FUNCTION_BLOCK FB_E2408_Manager
VAR_INPUT
	sendMessage			:ST_Modbus_Send_Frame;
END_VAR
VAR_OUTPUT
	bWriteError			:BOOL; 
	bReadError			:BOOL;
	bSendBufferusFull	:BOOL;
	bConnectError 		: BOOL;
	
	RData_Module_1	:ST_E2408_Data;
	RData_Module_2	:ST_E2408_Data;
	RData_Module_3	:ST_E2408_Data;
	RData_Module_4	:ST_E2408_Data;
	RData_Module_5	:ST_E2408_Data;
	RData_Module_6	:ST_E2408_Data;
END_VAR
VAR
	fbModbus_Master		:ModbusRtuMasterV2_KL6x22B;
	ReconnectTon		:TON;
	DataReadTon			:TON;
	bWriteExecute		:BOOL;
	bReadExecute		:BOOL;
	arrReceivedBuffer 	:ARRAY [0..200] OF WORD;
	arrSendBuffer 		:ARRAY [0..99] OF WORD;
	
	nModbusRead_Start_ADDR	:WORD;
	nModbusWrite_Start_ADDR	:WORD;
	nReadExecuteCount		:UDINT;
		
	fbStructModbusSend:FB_MODBUS_SEND_FIFO;
	stOutput:ST_MODBUS_SEND_FRAME;
	
	nWriteQuantity		:WORD;
	fallEdge			:F_TRIG;
	backCount			: UDINT;
	nCycle				: UDINT;
	ReceivedTime		: UDINT;
	ResendTon			: Ton;
	rinedge				: R_TRIG;
	WriteCount			: INT;
	CheckLoad			: REAL;
	ErrorCount			: INT;
	BufferCount_Zefo	: INT;
	fTrigWriteComplete	: F_TRIG;
	ReReadTon: TON;
	ReReadTrig			: BOOL;
	
	ReadInputRegsBusy		: BOOL;
	ReadInputRegsError		: BOOL;
	WriteSingleRegisterBusy	: BOOL;
	WriteSingleRegisterError: BOOL;
END_VAR

IF  ReadInputRegsError =FALSE THEN
	_Case();
	_CheckSendData();
ELSE
	ReconnectTon(IN:=ReconnectTon.Q=FALSE AND TRUE,pt:=T#1S);
	
	IF ReconnectTon.Q THEN
		
		ErrorCount := ErrorCount +1;
		
		IF ReadInputRegsError = TRUE THEN
			bReadExecute:=NOT bReadExecute;
		END_IF
		
	END_IF
END_IF

_ModbusFunction();
fbStructModbusSend();

bConnectError:= ReadInputRegsError;

ACTION _Case:
IF ReadInputRegsBusy = TRUE OR ReadInputRegsError = TRUE AND bWriteExecute = FALSE AND WriteSingleRegisterBusy = FALSE  THEN
	bReadExecute := FALSE;
	IF ReadInputRegsError = TRUE THEN
		bReadError:=TRUE;
	END_IF
END_IF

(*Copy Data*)
IF (ReadInputRegsBusy = FALSE AND ReadInputRegsError = FALSE)  THEN
	IF (fbModbus_Master.cbRead >0)  (*AND (arrReceivedBuffer[4] <> 0)*) THEN
		
	IF arrReceivedBuffer[4] = 0 THEN
		BufferCount_Zefo:=BufferCount_Zefo +1 ; 
	END_IF

		CASE nReadExecuteCount OF
			1:MEMCPY(ADR(RData_Module_1),ADR(arrReceivedBuffer),SIZEOF(RData_Module_1));
				ReceivedTime :=nCycle;
				nCycle:=0;
			2:MEMCPY(ADR(RData_Module_2),ADR(arrReceivedBuffer),SIZEOF(RData_Module_2));
			3:MEMCPY(ADR(RData_Module_3),ADR(arrReceivedBuffer),SIZEOF(RData_Module_3));
			4:MEMCPY(ADR(RData_Module_4),ADR(arrReceivedBuffer),SIZEOF(RData_Module_4));
			5:MEMCPY(ADR(RData_Module_5),ADR(arrReceivedBuffer),SIZEOF(RData_Module_5));
			6:MEMCPY(ADR(RData_Module_6),ADR(arrReceivedBuffer),SIZEOF(RData_Module_6));
		END_CASE
	END_IF
	
END_IF
nCycle:=nCycle+1;

(*Change Address*)
IF ReadInputRegsBusy = FALSE  AND ReadInputRegsError = FALSE  AND fbStructModbusSend.nBufferCount = 0 AND bWriteExecute = FALSE AND WriteSingleRegisterBusy = FALSE THEN
DataReadTon(IN:=TRUE,pT:=T#100MS);
	IF DataReadTon.Q THEN
		
		nReadExecuteCount:=nReadExecuteCount+1;
		DataReadTon(IN:=FALSE);
		bReadExecute:=TRUE;
		
		CASE nReadExecuteCount OF
			1:
				nModbusRead_Start_ADDR:=1;
			2:
				nModbusRead_Start_ADDR:=2;
			3:
				nModbusRead_Start_ADDR:=3;
			4:
				nModbusRead_Start_ADDR:=4;
			5:
				nModbusRead_Start_ADDR:=5;
			6:
				nModbusRead_Start_ADDR:=6;
			
				nReadExecuteCount:=0;
		ELSE
			nReadExecuteCount:=0;
			bReadExecute:=false;
		END_CASE
	END_IF
END_IF
END_ACTION

ACTION _CheckSendData:
IF WriteSingleRegisterBusy = FALSE OR WriteSingleRegisterError = TRUE THEN
	bWriteExecute := FALSE;
END_IF

IF fbStructModbusSend.nBufferCount > 0 AND bWriteExecute = FALSE AND WriteSingleRegisterBusy = FALSE THEN
	ResendTon(IN:=TRUE,pt:=T#150MS);
	rinedge(CLK:=ResendTon.Q);
	IF rinedge.q THEN
		ResendTon(IN:=FALSE);
		fbStructModbusSend.A_Remove(stOutput=>stOutput);
		
		nWriteQuantity:=stOutput.sendQuantity;
		nModbusWrite_Start_ADDR:=stOutput.StartAddress;
		MEMCPY(ADR(arrSendBuffer),ADR(stoutput.SendData),SIZEOF(stoutput.SendData));
		
		bWriteExecute:=TRUE;
		nReadExecuteCount:=0;
		rinedge(CLK:=FALSE);
		ReReadTrig:=FALSE;
	END_IF
END_IF
END_ACTION

ACTION _ModbusFunction:
//Write the Regs to Modbus Server Function16
IF ReadInputRegsBusy = FALSE THEN
	fbModbus_Master.WriteSingleRegister(
		UnitID:= 1, 
		Quantity:= nWriteQuantity, 
		MBAddr:= nModbusWrite_Start_ADDR, 
		cbLength:= SIZEOF(arrSendBuffer),
		pMemoryAddr:= ADR(arrSendBuffer),
		AuxQuantity:= , 
		AuxMBAddr:= , 
		AuxcbLength:= , 
		pAuxMemoryAddr:= , 
		Execute:= bWriteExecute,
		Timeout:= T#1S , 
		BUSY=>WriteSingleRegisterBusy ,
		Error=>WriteSingleRegisterError , 
		ErrorId=> , 
		cbRead=> );
END_IF

IF WriteSingleRegisterError THEN
	WriteCount:=WriteCount+1;
END_IF

IF WriteSingleRegisterBusy = FALSE THEN
	//Read the Regs FROM Modbus Server Function3
	fbModbus_Master.ReadInputRegs(
		UnitID:= 1, // 온도 콘트롤러 ID 
		Quantity:= 20, // 통신 데이터 사이즈
		MBAddr:= nModbusRead_Start_ADDR, //레지스터 주소
		cbLength:= SIZEOF(arrReceivedBuffer), 
		pMemoryAddr:= ADR(arrReceivedBuffer),
		AuxQuantity:= , 
		AuxMBAddr:= , 
		AuxcbLength:= , 
		pAuxMemoryAddr:= , 
		Execute:= bReadExecute,
		Timeout:= T#1S , 
		BUSY=>ReadInputRegsBusy ,
		Error=> ReadInputRegsError,
		ErrorId=> , 
		cbRead=> );		
END_IF
END_ACTION

ACTION _SendModbusCommand:
IF fbStructModbusSend.nLoad < 90THEN
	IF 	fbStructModbusSend.nLoad > CheckLoad THEN 
		CheckLoad := fbStructModbusSend.nLoad;
	END_IF
	
	fbStructModbusSend.A_Add(stinput:=sendMessage);	
END_IF
END_ACTION

END_FUNCTION_BLOCK

(* stored: Version 1.1.0.1
   POU FB_E2408_Manager: Id {9702cd75-241a-4a7b-8f90-3e54f3c6c47f}, SpecialFunc None
   Action _Case: Id {b5e5e4e6-f09c-4735-a18d-50cd827ec56f}
   Action _CheckSendData: Id {6562381a-d445-4f0c-9454-ad66b3a8766d}
   Action _ModbusFunction: Id {4fa7b19f-847a-46ef-a73f-4c96a6f0414c}
   Action _SendModbusCommand: Id {b19bf173-4bfe-4c73-b1c5-bae5c5bfcd31} *)
